FUNCTION_BLOCK FB_EnableDevice 
VAR_IN_OUT
	bTrigger			: BOOL;
END_VAR
VAR_INPUT
	sNetID				: T_AmsNetId;
	nSlaveAddr			: UINT;
END_VAR
VAR_OUTPUT
	bFinished			: BOOL;
	bSuccess			: BOOL;
END_VAR
VAR
	eState				: (WAIT_FOR_TRIGGER, SHUTDOWN, SWITCH_ON);
	tWait1				: TON;
	tWait2				: TON;
	fbGetStatusword		: FB_EcCoeSdoRead;
	nStatusword			: UINT;
	bGetStatusword		: BOOL;
	bExecuteTimer		: BOOL;
END_VAR

CASE eState OF
	WAIT_FOR_TRIGGER:
		IF bTrigger THEN
			bExecuteTimer	:= FALSE;
			bSuccess := TRUE;
			bFinished := FALSE;
			bTrigger := FALSE;
			eState := SHUTDOWN;
		END_IF
	
	SHUTDOWN:
		MAIN.Controlword.0 := 0;
		MAIN.Controlword.1 := 1;
		MAIN.Controlword.2 := 1;
		MAIN.Controlword.7 := 0;

		tWait1(PT := T#125MS,
			IN := bExecuteTimer);
			bExecuteTimer := TRUE;
		IF tWait1.Q THEN
			bExecuteTimer := FALSE;
			tWait2(IN := bGetStatusword,
				PT := T#250MS);
			fbGetStatusword(sNetId := sNetId,
				nSlaveAddr := nSlaveAddr,
				nIndex := 16#6041,
				nSubIndex := 0,
				pDstBuf := ADR(nStatusword),
				cbBufLen := SIZEOF(nStatusword),
				bExecute := bGetStatusword);
			bGetStatusword := TRUE;
			IF tWait2.Q THEN
				ADSLOGSTR(msgCtrlMask := ADSLOG_MSGTYPE_HINT,
					msgFmtStr := 'Shutdown',
					strArg := '');
				bExecuteTimer := FALSE;
				IF (nStatusword.0 = 1 AND nStatusword.5) 
					AND NOT (nStatusword.1 AND nStatusword.2 AND nStatusword.3
						AND nStatusword.6) THEN
 					eState := SWITCH_ON;
				ELSE 
					bSuccess := FALSE;
					bFinished := TRUE;
					eState := WAIT_FOR_TRIGGER;
				END_IF
			END_IF
		END_IF
		
	SWITCH_ON:
		ADSLOGSTR(msgCtrlMask := ADSLOG_MSGTYPE_HINT,
			msgFmtStr := 'Switch On',
			strArg := '');
		MAIN.Controlword.0 := 1;
		MAIN.Controlword.1 := 1;
		MAIN.Controlword.2 := 1;
		Main.Controlword.3 := 1;
		Main.Controlword.7 := 0;
		bExecuteTimer := TRUE;
		bGetStatusWord := TRUE;
		IF tWait1.Q THEN
			bExecuteTimer	:= FALSE;
			IF tWait2.Q THEN
				bGetStatusword := FALSE;
				IF nStatusword.0 AND nStatusword.1 AND nStatusword.5 
						AND NOT (nStatusword.2 AND nStatusword.3 AND nStatusword.6) THEN
					bSuccess := FALSE;
				END_IF
				bFinished := TRUE;
				eState := WAIT_FOR_TRIGGER;
			END_IF
		END_IF
END_CASE

END_FUNCTION_BLOCK

(* stored: Version 1.1.0.1, ProductVersion 3.1.4024.11
   POU FB_EnableDevice: Id {a410285a-0c2f-47a6-bfb6-f23d8e315db6}, SpecialFunc None *)
